FUNCTION IsRoiSizeOK_Dint : BOOL
VAR_INPUT
    RoiRectangle : TcVnRectangle_DINT;
    ImageWidth : UDINT;
    ImageHeight : UDINT;
END_VAR
VAR
    width : DINT;
    height : DINT;
END_VAR

IF NOT TryConvert_UDINT_TO_DINT(ImageWidth, width) THEN
    RETURN;
END_IF

IF NOT TryConvert_UDINT_TO_DINT(ImageHeight, height) THEN
    RETURN;
END_IF

IF NOT (RoiRectangle.nX < width) THEN
	RETURN;
END_IF

IF NOT (RoiRectangle.nY < height) THEN
	RETURN;
END_IF

IF NOT (RoiRectangle.nWidth <= (width - RoiRectangle.nX)) THEN
	RETURN;
END_IF

IF NOT (RoiRectangle.nHeight <= (height - RoiRectangle.nY)) THEN
	RETURN;
END_IF

IsRoiSizeOK_Dint := TRUE;

END_FUNCTION

(* stored: Version 1.1.0.1, ProductVersion 3.1.4026.13
   POU IsRoiSizeOK_Dint: Id {96080696-cb86-0eb9-15ba-3c04f533f819}, SpecialFunc None *)
